// TIA Portal V17 export
// export: Created 2023-02-25T15:48:31.0242205Z, ExportSetting WithDefaults, DisplayName Totally Integrated Automation Portal, DisplayVersion V17, DisplayName TIA Portal Openness, DisplayVersion V17, DisplayName TIA Portal Version Control Interface, DisplayVersion V17, DisplayName TIA Portal Test Suite Advanced, DisplayVersion V17, DisplayName STEP 7 Professional, DisplayVersion V17, DisplayName SIMATIC Energy Suite, DisplayVersion V17, DisplayName STEP 7 Safety, DisplayVersion V17, DisplayName WinCC Professional, DisplayVersion V17
DATA_BLOCK "LOG_AutoControle_DB"   // DB11
VERSION : 0.1
// stored: AutoNumber true, InstanceOfName LOG_AutoControle, InstanceOfType FB
"LOG_AutoControle"
   // VAR_INPUT
   //    StartLine : Bool;
   //    StopLine : Bool;
   //    AutoMode : Bool;
   //    SmallPackage : Bool;
   //    MediumPackage : Bool;
   //    LargePackage : Bool;
   //    D3 : Bool;
   //    D4 : Bool;
   //    D5 : Bool;
   //    D6 : Bool;
   //    FirstScan : Bool;
   // END_VAR
   // VAR_OUTPUT
   //    ConveyorsAuto : "stt_Conveyor";
   // END_VAR
   // VAR
   //    s1 : Bool;
   //    s2 : Bool;
   //    s3 : Bool;
   //    s4 : Bool;
   //    s5 : Bool;
   //    P_D3_1 : Bool;
   //    P_D3_2 : Bool;
   //    P_D3_3 : Bool;
   //    N_D4 : Bool;
   //    N_D5 : Bool;
   //    N_D6 : Bool;
   // END_VAR
BEGIN
END_DATA_BLOCK
